{attribute 'pack_mode' := '1'}
TYPE ST_ReadCellData :
STRUCT
	stReadListReturnInfo		: ARRAY [1..1] OF ST_UAReadListReturnInfo;
	stCell						: ST_StatusCell;

END_STRUCT
END_TYPE

(* stored: Version 1.1.0.1, ProductVersion 3.1.4024.5
   DUT ST_ReadCellData: Id {46146e78-8c60-484a-820b-e21bd5ad9ba4} *)
